Staubli VAL3: here.pgx

public program here()
begin
  saveData:rif2=here(saveData:tData[0].tcp,world)
  saveData:bCheck=true
end
